// TIA Portal project "modbus_rs485" (V15)

(* hardware
DEVICE "S7-1200 station_1"  S7-1200 Station
   slot 0: "Rack_0"  S7-1200 Rack  Rack  V1.0
   slot 1: "PLC_1"  CPU 1214C DC/DC/DC  6ES7 214-1AG40-0XB0  V4.0
   slot 101: "CM 1241 (RS422/485)_1"  6ES7 241-1CH32-0XB0  V2.0
*)

// ===== PLC "PLC_1"  CPU 1214C DC/DC/DC =====

VAR_GLOBAL   // PLC tag table "Default tag table"
   "System_Byte" AT %MB1 : Byte;
   "FirstScan" AT %M1.0 : Bool;
   "DiagStatusUpdate" AT %M1.1 : Bool;
   "AlwaysTRUE" AT %M1.2 : Bool;
   "AlwaysFALSE" AT %M1.3 : Bool;
   "Clock_Byte" AT %MB0 : Byte;
   "Clock_10Hz" AT %M0.0 : Bool;
   "Clock_5Hz" AT %M0.1 : Bool;
   "Clock_2.5Hz" AT %M0.2 : Bool;
   "Clock_2Hz" AT %M0.3 : Bool;
   "Clock_1.25Hz" AT %M0.4 : Bool;
   "Clock_1Hz" AT %M0.5 : Bool;
   "Clock_0.625Hz" AT %M0.6 : Bool;
   "Clock_0.5Hz" AT %M0.7 : Bool;
   "Tag_1" AT %M20.0 : Bool;
   "Tag_2" AT %M30.0 : Bool;
   "step" AT %M5.0 : Bool;
   "Gap vat" AT %M60.0 : Bool;
   "Nha vat" AT %M70.0 : Bool;
END_VAR

DATA_BLOCK "Data_block_1"   // DB3
{ S7_Optimized_Access := 'FALSE' }
VERSION : 0.1
   VAR
      Data_Trans : Word;
   END_VAR
BEGIN
END_DATA_BLOCK

// folder: System blocks/Program resources

DATA_BLOCK "IEC_Timer_0_DB"   // DB4
{ S7_Optimized_Access := 'TRUE' }
AUTHOR : Simatic
FAMILY : IEC
NAME : IEC_TMR
VERSION : 1.0
// stored: InstanceOfName IEC_TIMER
"IEC_TIMER"
BEGIN
END_DATA_BLOCK

DATA_BLOCK "IEC_Timer_0_DB_1"   // DB5
{ S7_Optimized_Access := 'TRUE' }
AUTHOR : Simatic
FAMILY : IEC
NAME : IEC_TMR
VERSION : 1.0
// stored: InstanceOfName IEC_TIMER
"IEC_TIMER"
BEGIN
END_DATA_BLOCK

// folder: (top level)

ORGANIZATION_BLOCK "Main"   // OB1, LAD, ProgramCycle
TITLE = "Main Program Sweep (Cycle)"
{ S7_Optimized_Access := 'TRUE' }
VERSION : 0.1
   VAR_INPUT
      Initial_Call : Bool;   // Initial call of this OB
      Remanence : Bool;   // =True, if remanent data are available
   END_VAR
BEGIN

REGION Network 1
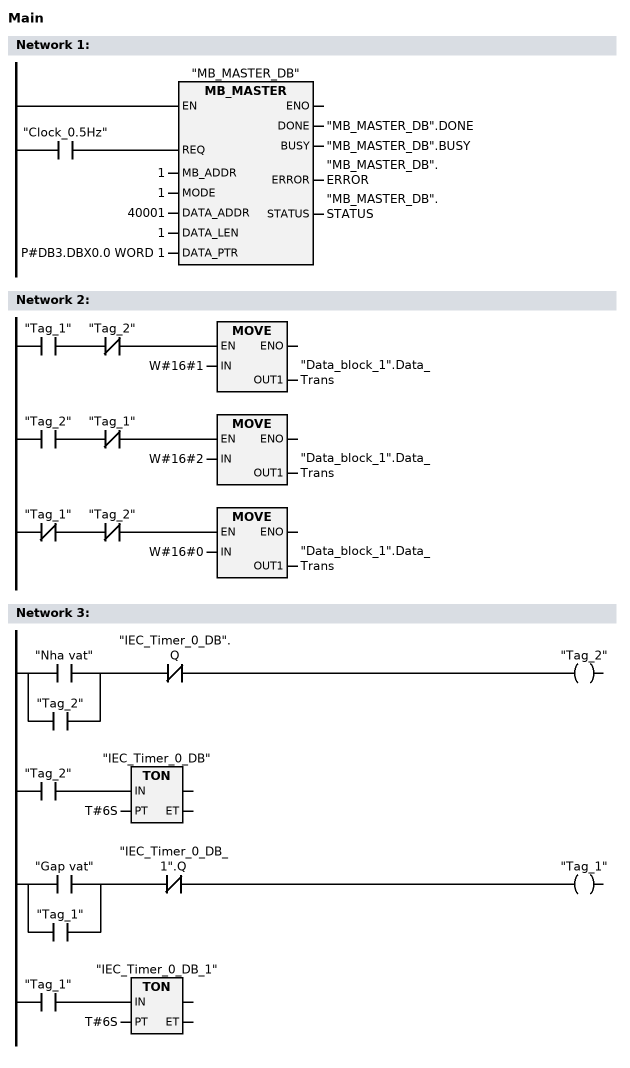
   "MB_MASTER_DB"(REQ := "Clock_0.5Hz",   // MB_MASTER
                  MB_ADDR := 1,
                  MODE := 1,
                  DATA_ADDR := 40001,
                  DATA_LEN := 1,
                  DATA_PTR := P#DB3.DBX0.0 WORD 1,
                  DONE => "MB_MASTER_DB".DONE,
                  BUSY => "MB_MASTER_DB".BUSY,
                  ERROR => "MB_MASTER_DB".ERROR,
                  STATUS => "MB_MASTER_DB".STATUS);
END_REGION

REGION Network 2
   RUNG wire#powerrail
      Contact( "Tag_1" )
      I_Contact( "Tag_2" )
      Move(in := W#16#1, out1 => "Data_block_1".Data_Trans)
   END_RUNG
   RUNG wire#powerrail
      Contact( "Tag_2" )
      I_Contact( "Tag_1" )
      Move(in := W#16#2, out1 => "Data_block_1".Data_Trans)
   END_RUNG
   RUNG wire#powerrail
      I_Contact( "Tag_1" )
      I_Contact( "Tag_2" )
      Move(in := W#16#0, out1 => "Data_block_1".Data_Trans)
   END_RUNG
   // the same network as SCL:
   IF "Tag_1" AND NOT "Tag_2" THEN "Data_block_1".Data_Trans := W#16#1; END_IF;
   IF "Tag_2" AND NOT "Tag_1" THEN "Data_block_1".Data_Trans := W#16#2; END_IF;
   IF NOT "Tag_1" AND NOT "Tag_2" THEN "Data_block_1".Data_Trans := W#16#0; END_IF;
END_REGION

REGION Network 3
   "Tag_2" := ("Nha vat" OR "Tag_2") AND NOT "IEC_Timer_0_DB".Q;
   "IEC_Timer_0_DB".TON(IN := "Tag_2", PT := T#6S);
   "Tag_1" := ("Gap vat" OR "Tag_1") AND NOT "IEC_Timer_0_DB_1".Q;
   "IEC_Timer_0_DB_1".TON(IN := "Tag_1", PT := T#6S);
END_REGION
END_ORGANIZATION_BLOCK

ORGANIZATION_BLOCK "Startup"   // OB100, LAD, Startup
TITLE = "Complete Restart"
{ S7_Optimized_Access := 'TRUE' }
VERSION : 0.1
   VAR_INPUT
      LostRetentive : Bool;   // True if retentive data are lost
      LostRTC : Bool;   // True if date and time are lost
   END_VAR
BEGIN

REGION Network 1
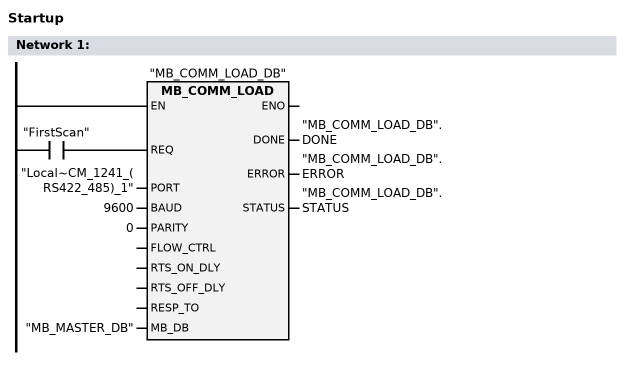
   "MB_COMM_LOAD_DB"(REQ := "FirstScan",   // MB_COMM_LOAD
                     PORT := "Local~CM_1241_(RS422_485)_1",
                     BAUD := 9600,
                     PARITY := 0,
                     MB_DB := "MB_MASTER_DB",
                     DONE => "MB_COMM_LOAD_DB".DONE,
                     ERROR => "MB_COMM_LOAD_DB".ERROR,
                     STATUS => "MB_COMM_LOAD_DB".STATUS);
END_REGION
END_ORGANIZATION_BLOCK